FUNCTION_BLOCK TurnTableControllerIReq (* Turn Table Controller Interface Requier *)
  (* Standard: 61499-2 *)
  (* Version 0.2, 2003-12-05, JHC, Rockwell Automation, Renamed from NEWCOMPFB. *)
  (* Version 0.1, 2002-01-08, JHC, Rockwell Automation, Added DLY FB as example. *)
  (* Version 0.0, 2000-05-27, JHC, Rockwell Automation *)
  (* Compiler header: package fb.rt.dasdA1.A2.TurnTable; *)
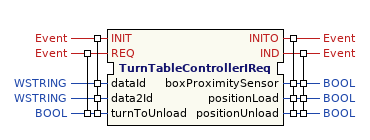
  EVENT_INPUT
    INIT WITH dataId, data2Id, turnToUnload; (* Initialization Request *)
    REQ WITH turnToUnload;
  END_EVENT
  EVENT_OUTPUT
    INITO WITH boxProximitySensor, positionLoad, positionUnload; (* Initialization Confirm *)
    IND WITH boxProximitySensor, positionLoad, positionUnload;
  END_EVENT
  VAR_INPUT
    dataId : WSTRING;
    data2Id : WSTRING;
    turnToUnload : BOOL;
  END_VAR
  VAR_OUTPUT
    boxProximitySensor : BOOL;
    positionLoad : BOOL;
    positionUnload : BOOL;
  END_VAR
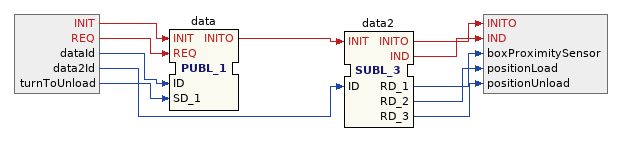
  FBS
    data : PUBL_1;
    data2 : SUBL_3;
  END_FBS
  EVENT_CONNECTIONS
    INIT TO data.INIT;
    REQ TO data.REQ;
    data.INITO TO data2.INIT;
    data2.INITO TO INITO;
    data2.IND TO IND;
  END_CONNECTIONS
  DATA_CONNECTIONS
    dataId TO data.ID;
    turnToUnload TO data.SD_1;
    data2Id TO data2.ID;
    data2.RD_1 TO boxProximitySensor;
    data2.RD_2 TO positionLoad;
    data2.RD_3 TO positionUnload;
  END_CONNECTIONS
END_FUNCTION_BLOCK
